(* PLC project SafeLOGIC, BrAutomation SafeDESIGNER  5.24.1.0 *)
(* stored: companyURL http://www.br-automation.com, creationDateTime Fri Nov 28 15:05:03 2025 *)

PROGRAM DI_MON
  VAR  (* added by the conversion: wires and edge detectors of the diagram *)
    _AND_S11_OUT : ANY;
  END_VAR

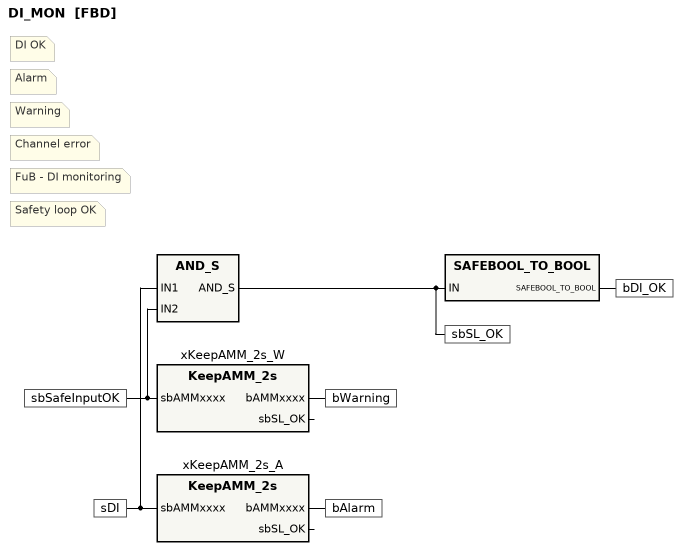
(* FBD diagram, written out as Structured Text *)
(* FuB - DI monitoring *)
(* Alarm *)
xKeepAMM_2s_A(sbAMMxxxx := sDI);
bAlarm := xKeepAMM_2s_A.bAMMxxxx;
(* Safety loop OK *)
(* DI OK *)
_AND_S11_OUT := AND_S(sDI, sbSafeInputOK);
bDI_OK := SAFEBOOL_TO_BOOL(_AND_S11_OUT);
sbSL_OK := _AND_S11_OUT;
(* Channel error *)
(* Warning *)
xKeepAMM_2s_W(sbAMMxxxx := sbSafeInputOK);
bWarning := xKeepAMM_2s_W.bAMMxxxx;
END_PROGRAM
